VAR_GLOBAL
	ads_watch_dog	:	FB_ADS_WATCHDOG;
END_VAR

(* stored: Version 1.1.0.1, ProductVersion 3.1.4024.2
   GVL GVL_VAC_INTF: Id {53b9bff0-0c14-4179-9583-15209156ddbc} *)
